FUNCTION_BLOCK FB_GroupElement_HMI EXTENDS FB_BaseGroupElement_HMI IMPLEMENTS ITF_Component_HMI
VAR
	itfGroupElementConnector			: ITF_GroupElement_HMI_Connector;
	refstGroupElementData				: REFERENCE TO ST_GroupElement_HMI;
END_VAR

METHOD FB_init : BOOL
VAR_INPUT
	bInitRetains : BOOL; // if TRUE, the retain variables are initialized (warm start / cold start)
	bInCopyCode : BOOL;  // if TRUE, the instance afterwards gets moved into the copy code (online change)
	itfBaseLoggerConnector				: ITF_BaseLogger_HMI_Connector;	//bezpośredni łącznik do logera
	itfGroupElementConnector			: ITF_GroupElement_HMI_Init;
END_VAR
//Przypisanie do elementu który własnie stworzyliśmy
THIS^.itfGroupElementConnector			:= itfGroupElementConnector;
//Przypisanie do elementów z biblioteki
THIS^.itfBaseLoggerElementConnector		:= itfGroupElementConnector;
THIS^.itfBaseComponentConnector			:= itfGroupElementConnector;
THIS^.itfBaseControlElementConnector	:= itfGroupElementConnector;
THIS^.itfBaseGroupElementConnector		:= itfGroupElementConnector;
//
THIS^.itfBaseLoggerConnector			:= itfBaseLoggerConnector;

IF (THIS^.itfGroupElementConnector <> 0 AND
	THIS^.itfBaseLoggerElementConnector <> 0 AND
	THIS^.itfBaseComponentConnector	<> 0 AND
	THIS^.itfBaseControlElementConnector <> 0 AND
	THIS^.itfBaseGroupElementConnector <> 0 AND
	THIS^.itfBaseLoggerConnector <> 0) THEN
	THIS^.bIsInit						:= TRUE;
END_IF
END_METHOD

END_FUNCTION_BLOCK

(* stored: Version 1.1.0.1, ProductVersion 3.1.4024.15
   POU FB_GroupElement_HMI: Id {19883d18-afce-4591-ab72-0deda3f3642e}, SpecialFunc None
   Method FB_init: Id {60cf9aa3-a3c1-477d-943b-0793fbe6bf08} *)
